FUNCTION_BLOCK INTERNAL FINAL FB_TestFixed32Message IMPLEMENTS I_Message
VAR
    fbMessageParser : FB_MessageParser(ipMessage:= THIS^);
    fbMessageWriter : FB_MessageWriter(ipMessage:= THIS^);
    nValue : UDINT;
END_VAR

METHOD CalculateSize : UDINT
VAR_INPUT
END_VAR
CalculateSize := F_ComputeTagSize(1) + SIZEOF(nValue);
END_METHOD

METHOD MergeFrom : HRESULT
VAR_IN_OUT
    fbParseCtx : FB_ParseContext;
END_VAR
VAR
    nTag : UDINT;
END_VAR
REPEAT
MergeFrom := fbParseCtx.ReadTag(nTag=> nTag);
IF SUCCEEDED(MergeFrom) AND nTag = 0 THEN
    EXIT;
END_IF

IF FAILED(MergeFrom) THEN
    RETURN;
END_IF

CASE nTag OF
    16#0D:
        MergeFrom := fbParseCtx.ReadFixed32(nValue=> nValue);
ELSE
    MergeFrom := fbParseCtx.SkipLastField();
END_CASE
UNTIL FAILED(MergeFrom) OR nTag = 0
END_REPEAT
END_METHOD

PROPERTY MessageValue : T_Any
GET
MessageValue := F_ToAnyType(anyArg:= nValue);
END_GET
END_PROPERTY

PROPERTY Parser : REFERENCE TO FB_MessageParser
GET
Parser REF= fbMessageParser;
END_GET
END_PROPERTY

PROPERTY Writer : REFERENCE TO FB_MessageWriter
GET
Writer REF= fbMessageWriter;
END_GET
END_PROPERTY

METHOD WriteTo : HRESULT
VAR_IN_OUT
    fbWriteCtx : FB_WriteContext;
END_VAR
WriteTo := fbWriteCtx.WriteTag(1, E_WireType.Fixed32);
IF FAILED(WriteTo) THEN
    RETURN;
END_IF

WriteTo := fbWriteCtx.WriteFixed32(nValue);
END_METHOD

END_FUNCTION_BLOCK

(* stored: Version 1.1.0.1
   POU FB_TestFixed32Message: Id {88505a11-3a8b-4d3a-86c7-667689b26c36}, SpecialFunc None
   Method CalculateSize: Id {b385b862-57ca-4a13-81af-1fdb807a2199}
   Method MergeFrom: Id {913f0298-d0f1-434f-931d-6f2eb2a1f843}
   Property MessageValue: Id {12079bee-53ff-4ec9-863c-dfe11761c510}
   Get Get: Id {04919680-96df-41dc-ac89-25ff2c4dde1b}
   Property Parser: Id {d6b0d26a-48f6-4e94-8643-52afe2fcb7a4}
   Get Get: Id {f7504f09-5125-4e78-898b-a961d7e3383f}
   Property Writer: Id {2df17427-080e-4e2c-a02b-2f2d7dfb8254}
   Get Get: Id {03e5638e-9d70-4165-8af2-0a6cfc1fd60c}
   Method WriteTo: Id {842e8dd1-ccfb-42bc-9bbf-b4ebf860310f} *)
